PROGRAM Pedal
VAR
	
END_VAR

END_PROGRAM

(* stored: Version 1.1.0.1, ProductVersion 3.1.4024.3
   POU Pedal: Id {b480e77f-b772-4b6b-8c1b-2f16ad405884}, SpecialFunc None *)
